FUNCTION_BLOCK F_ADD_DT_TIME (* Adds two number values *)
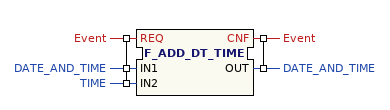
  EVENT_INPUT
    REQ WITH IN1, IN2; (* Normal Execution Request *)
  END_EVENT
  EVENT_OUTPUT
    CNF WITH OUT; (* Execution Confirmation *)
  END_EVENT
  VAR_INPUT
    IN1 : DATE_AND_TIME; (* First funtion input *)
    IN2 : TIME; (* Second function input *)
  END_VAR
  VAR_OUTPUT
    OUT : DATE_AND_TIME; (* Function output *)
  END_VAR
END_FUNCTION_BLOCK
